        |     # rotate 180 degrees about x. then rotate (90 deg + heading1 degrees) about z ccw
        |     m1 = get_rotation_matrix_from_description("x", -1, 180 * pi / 180)
        |     m2 = get_rotation_matrix_from_description("z", 1, heading1 + pi/2)
        |     m3 = multiply_matrix(m2, m1) #we rotate m1 first then m2, so we multiply in backwards order: 2 then 1
        |     rxryrz2 = convert_matrix_to_axang(m3)
        |     rx2 = rxryrz2[0]
        |     ry2 = rxryrz2[1]
        |     rz2 = rxryrz2[2]
        | 
        |     # calculate point centerchamfers (where the center of the two chamfers intersect
        |     pcx = x0 + (leftwallthickmm + deepchambumpmm) * l1delxunit + (rightwallthickmm + deepchambumpmm) * l2delxunit
        |     pcy = y0 + (leftwallthickmm + deepchambumpmm) * l1delyunit + (rightwallthickmm + deepchambumpmm) * l2delyunit
        |     pcz = z0
        | 
        |     # calculate point1 (start of weld)
        |     p1x = pcx + l2delxunit * wd1
        |     p1y = pcy + l2delyunit * wd1
        |     p1z = pcz
        |     point1 = p[p1x, p1y, p1z, rx1, ry1, rz1]
        | 
        |     # calculate point2 (end of segment 1)
        |     p2x = pcx
        |     p2y = pcy
        |     p2z = pcz
        |     point2 = p[p2x, p2y, p2z, rx1, ry1, rz1]
        | 
        |     # calculate point3 (point at end of turn)
        |     slide = 0.00 # slide distance : the distance the tip slides forward as it turns
        |     p3x = pcx + slide * l1delxunit
        |     p3y = pcy + slide * l1delyunit
        |     p3z = pcz
        |     point3 = p[p3x, p3y, p3z, rx2, ry2, rz2]
        | 
        |     # calculate point4 (end of segment 2)
        |     p4x = pcx + wd2 * l1delxunit
        |     p4y = pcy + wd2 * l1delyunit
        |     p4z = pcz
        |     point4 = p[p4x, p4y, p4z, rx2, ry2, rz2]
        | 
        |     # third path
        | 
        |     # calculate rxryrz3 (gun pointing down, preheat pointing toward corner. for right seam, pointing right)
        |     # start with rxryrz = 0,0,0 (gun facing up, preheat facing y+ axis.
        |     # rotate it 180 degrees about x axis. gun facing down, preheat facing y- axis
        |     # rotate it about 135 degrees ccw about z axis. x+ to heading3 is about 225 degrees. so our angle is heading3 - 90 degrees
        |     m1 = get_rotation_matrix_from_description("x", -1, 180 * pi / 180) # rotation 1: 180 degrees forward about x axis
        |     m2 = get_rotation_matrix_from_description("z", 1, heading3 - pi/2) # rotation 2
        |     m3 = multiply_matrix(m2, m1) #we rotate m1 first then m2, so we multiply in backwards order: 2 then 1
        |     rxryrz3 = convert_matrix_to_axang(m3)
        |     rx3 = rxryrz3[0]
        |     ry3 = rxryrz3[1]
        |     rz3 = rxryrz3[2]
        | 
        |     # calculate rxryrz4 (gun at 45 around corner)
        |     m1 = get_rotation_matrix_from_description("x", -1, 135 * pi / 180) # rotation 1: 135 degrees forward about x axis
        |     m2 = get_rotation_matrix_from_description("z", 1, heading3 - pi/2)
        |     m3 = multiply_matrix(m2, m1) #we rotate m1 first then m2, so we multiply in backwards order: 2 then 1
        |     rxryrz4 = convert_matrix_to_axang(m3)
        |     rx4 = rxryrz4[0]
        |     ry4 = rxryrz4[1]
        |     rz4 = rxryrz4[2]
        | 
        |     # calculate rxryrz5 (gun straight into right seam side chamfer, preheat down)
        |     # rotate about x 90 (forward). then rotate about z ~ 135 (ccw)
        |     m1 = get_rotation_matrix_from_description("x", -1, 90 * pi / 180)
        |     m2 = get_rotation_matrix_from_description("z", 1, heading3 - pi/2)
        |     m3 = multiply_matrix(m2, m1) #we rotate m1 first then m2, so we multiply in backwards order: 2 then 1
        |     rxryrz5 = convert_matrix_to_axang(m3)
        |     rx5 = rxryrz5[0]
        |     ry5 = rxryrz5[1]
        |     rz5 = rxryrz5[2]
        | 
        |     # calculate rxryrz6 (gun straight into right seam side chamfer, preheat down, 10 degrees tiltback)
        |     tiltangledeg = 10 # ten degree angle of tilt
        |     m1 = get_rotation_matrix_from_description("x", -1, (90 + tiltangledeg) * pi / 180) # rotation 1: 135 degrees forward about x axis
        |     m2 = get_rotation_matrix_from_description("z", 1, heading3 - pi/2)
        |     m3 = multiply_matrix(m2, m1) #we rotate m1 first then m2, so we multiply in backwards order: 2 then 1
        |     rxryrz6 = convert_matrix_to_axang(m3)
        |     rx6 = rxryrz6[0]
        |     ry6 = rxryrz6[1]
        |     rz6 = rxryrz6[2]
        | 
        |     # calculate pointtopcham (the point at the top of the endwall chamfer) ( WHERE POINT3 WOULD BE IF RADIUS WAS 0)
        |     ptcx = x0 + leftwallthickmm * l1delxunit
        |     ptcy = y0 + leftwallthickmm * l1delyunit
        |     ptcz = z0
        | 
        |     # calculate point201 (weld start)
        |     # if deepchamfer, just ignore that. because if its deep chamfer then it filled more as well. so the hot extrudant should be to the same spot (same distance from the pointtopcham) whether it's big weld or small weld
        |     adjust = 0.0 # if you want to move the start point further away from corner (positive, mm) or closer to corner
        |     p201x = x0 + rightwallthickmm * l2delxunit + leftwallthickmm * l1delxunit + adjust * l2delxunit
        |     p201y = y0 + rightwallthickmm * l2delyunit + leftwallthickmm * l1delyunit + adjust * l2delyunit
        |     p201z = z0
        |     point201 = p[p201x, p201y, p201z, rx3, ry3, rz3]
        | 
        |     # the round over distance is the distance from pointbottomvcham to point2 (which will be the same as distance to p4)
        |     roundoverdistance = 0.05
        |     rod = roundoverdistance * 25.4 / 1000
        | 
        |     # calculate point202 (start of roundover)
        |     p202x = ptcx + rod * l2delxunit
        |     p202y = ptcy + rod * l2delyunit
        |     p202z = z0
        |     point202 = p[p202x, p202y, p202z, rx3, ry3, rz3]
        | 
        |     # calculate point203 (middle of roundover)
        |     # we know that the angle is exactly 90 degrees
        |     delta = calc_rod_midpoint_90deg(rod)
        |     p203z = ptcz - delta
        |     p203x = ptcx + delta * l2delxunit
        |     p203y = ptcy + delta * l2delyunit
        |     point203 = p[p203x, p203y, p203z, rx4, ry4, rz4]
        | 
        |     # calculate point204 (end of roundover)
        |     point204 = p[ptcx, ptcy, ptcz - rod, rx5, ry5, rz5]
        | 
        |     # calculate trail out points (tilt back and ride)
        |     botvcham = wd3 # where is the bottom of the v chamfer (z distance from top corner)
        |     tcpdiff = 14 # mm. the difference between backofhole tcp and welder tcp (tip)
        |     # point101 will still use backofhole, but points 102 and 103 will use normal weld tip tcp
        |     # calculate point5a (point101) (start of tilt back) (start of unflatten)
        |     dist = 1.5 * 25.4/1000 + tcpdiff/1000 # distance from botvcham
        |     p101x = ptcx
        |     p101y = ptcy
        |     p101z = ptcz - wd3 + dist
        |     point101 = p[p101x, p101y, p101z, rx5, ry5, rz5]
        | 
        |     # calculate point5b (point 102) (end of unflatten)
        |     dist = 0.5 * 25.4 / 1000
        |     tiltraise = 0.006
        |     p102x = ptcx + l2delxunit * tiltraise * -1
        |     p102y = ptcy + l2delyunit * tiltraise * -1
        |     p102z = ptcz - wd3 + dist
        |     point102 = p[p102x, p102y, p102z, rx6, ry6, rz6]
        | 
        |     # calculate point 5c (point 103) (end of smear)
        |     dist = -2 * 25.4/1000
        |     point103 = p[p102x, p102y, ptcz - wd3 + dist, rx6, ry6, rz6]
        | 
        |     # return
        |     struct2 = struct(point1=point1, point2=point2, point3=point3, point4=point4, point201=point201, point202=point202, point203=point203, point204=point204, point101=point101, point102=point102, point103=point103)
        |     return struct2
        | 
        | end
        | 
        | 
        | def main_calculate_cover_straight(p11, p12, p21, p22, sidewallthick, leftpoint, rightpoint, deepcovercham):
        |     struct1 = analyze_touchpoints_only_cover_straight(p11, p12, p21, p22, leftpoint)
        |     struct2 = calculate_straight_points_cover(struct1, sidewallthick, leftpoint, rightpoint, deepcovercham)
        |     #struct2 = calculate_DOtA_points_left_extended(struct1, list1, chamferover, chamferup, tcp_pose_top)
        |     #struct3 = check_validity_left(struct1, struct2)
        |     return struct2
        | 
        | end
        | 
        | # calculates the line of intersection of the sidewall plane (assumed vertical) and the cover plane (assumed perpendicular to sidewall plane)
        | # returns a struct containing point0 (point on the intersection line, same y as leftpoint) and 3 components of the unit vector left to right and 2 components of the other direction in 2d
        | def analyze_touchpoints_only_cover_straight(p11, p12, p21, p22, leftpoint):
        |     # calculate slope of sidewall in x-y plane
        |     # get the raw points from the first line
        |     l1p1x=p11[0]
        |     l1p1y=p11[1]
        |     l1p2x=p12[0]
        |     l1p2y=p12[1]
        | 
        |     # equate the first line in 2d space
        |     ml1 = (l1p2y-l1p1y) / (l1p2x-l1p1x)
        | 
        |     # b = y - mx
        |     bl1 = l1p1y - ml1 * l1p1x
        | 
        |     # calculate the cover plane
        |     # if two planes are perpendicular, then their normal vectors must be perpendicular.
        |     # the first planes normal vector is n1, which is taken from the equation of the plane ax + by + cz = d -> <a, b, c>
        |     # the second plane's normal vector is perpendicular to all vectors contained in the plane
        |     # p21 to p22 is a vector v contained within plane 2.
        |     # n2 is normal to both n1 AND v. to achieve a vector that is normal to both, take the cross product
        | 
        |     # plane 1 (y = mx + b) -> (b = -mx +1y +0z)
        |     n1 = [-1 * ml1, 1, 0]
        | 
        |     # v=P2−P1=(x2−x1,y2−y1,z2−z1)
        |     v = [p21[0]-p22[0], p21[1]-p22[1], p21[2]-p22[2]]
        | 
        |     #v n2 = cross product of n1 and v
        |     n2x = n1[1]*v[2] - n1[2]*v[1]
        |     n2y = n1[2]*v[0] - n1[0]*v[2]
        |     n2z = n1[0]*v[1] - n1[1]*v[0]
        |     n2 = [n2x, n2y, n2z]
        | 
        |     # find the d of the second plane
        |     # n2x * x + n2y * y + n2z * z = d0
        |     d = n2x * p21[0] + n2y * p21[1] + n2z * p21[2]
        | 
        |     # find the intersection line of the two planes
        |     # find the direction vector of that line by taking the cross product of the normal vector of those two planes
        |     v3x = n1[1]*n2[2] - n1[2]*n2[1]
        |     v3y = n1[2]*n2[0] - n1[0]*n2[2]
        |     v3z = n1[0]*n2[1] - n1[1]*n2[0]
        |     v3 = [v3x, v3y, v3z]
        | 
        |     # normalize the vector so the magnitude is 1
        |     magnitude2 = v3x * v3x + v3y * v3y + v3z * v3z
        |     magnitude = sqrt(magnitude2)
        |     v3xunit = v3x/magnitude
        |     v3yunit = v3y/magnitude
        |     v3zunit = v3z/magnitude
        | 
        |     # make sure it is going the right way (from left to right). make sure the v3yunit is positive
        |     if v3yunit < 0:
        |         v3xunit = v3xunit * -1
        |         v3yunit = v3yunit * -1
        |         v3zunit = v3zunit * -1
        |     end
        | 
        |     # next we have to find a point on the line by setting one of the dimensions and solving the system of equations
        |     # i will pick the y value of the left teach point
        |     y = leftpoint[1]
        |     # plane 1: -ml1 * x + 1 * y + 0 * z = bl1
        |     # -ml1 * x = bl1 - y
        |     x = (bl1 - y)/ (-1 * ml1)
        |     # plane 2: d = n2x * x + n2y * y + n2z * z
        |     # (d - n2x * x - n2y * y) = n2z * z
        |     z = (d - n2x * x - n2y * y) / n2z
        | 
        |     # make point0 into a pose
        |     point0 = p[x, y, z, 0, 0, 0]
        | 
        |     # find heading of main line
        |     heading1 = convert_uv_to_heading(v3xunit, v3yunit)
        | 
        |     # make a unit vector perpendicular to this one in the xy plane pointing x -. will be used to move over the chamfer distance
        |     ml2 = -1 / ml1
        |     # y = ml2 * x + unknownB
        |     # vector = [1, ml2]
        |     mag2 = 1 + ml2 * ml2
        |     mag = sqrt(mag2)
        |     v4xunit = 1 / mag
        |     v4yunit = ml2 / mag
        |     # switch is to the x direction is negative
        |     v4xunit = -1 * v4xunit
        |     v4yunit = -1 * v4yunit
        | 
        |     ret = struct(point0=point0, v3xunit=v3xunit, v3yunit=v3yunit, v3zunit=v3zunit, heading1=heading1, v4xunit=v4xunit, v4yunit=v4yunit)
        |     return ret
        | end
        | 
        | def calculate_straight_points_cover(struct1, sidewallthick, leftpointteach, rightpointteach, deepcovercham):
        |     # get the stuff
        |     point0 = struct1[0]
        |     p0x = point0[0]
        |     p0y = point0[1]
        |     p0z = point0[2]
        |     v3xunit = struct1[1]
        |     v3yunit = struct1[2]
        |     v3zunit = struct1[3]
        |     heading1 = struct1[4]
        |     v4xunit = struct1[5]
        |     v4yunit = struct1[6]
        |     sidewallthick = sidewallthick
        |     lpy = leftpointteach[1]
        |     rpy = rightpointteach[1]
        | 
        |     # first, check if we need a lift column raise
        |     # (we do, because for maximum reach we want to make the lift pedestal be even with the top of the covers)
        |     zpi = p0z
        |     if zpi > 0:
        |         liftcolumnzneeded = zpi * 1000.0 # the robot uses coordinates in meters, but the lift column uses coordinates in mm
        |         coverz = 0
        |     else:
        |         coverz = zpi
        |     end
        | 
        |     if deepcovercham:
        |         deepchambumpmm = 0.09 * 25.4/1000 # if there is a deep chamfer on the cover, bump the welder inwards 0.09 more inches.
        |     else:
        |         deepchambumpmm = 0.0
        |     end
        | 
        |     # calculate pointtopvcham
        |     chamferover = sidewallthick * 25.4 / 1000.0 + deepchambumpmm
        |     tiltraise = 0.006 # 6 mm raise needed for the tip to clear the plane during tiltback
        |     x = p0x + v4xunit * chamferover
        |     y = p0y + v4yunit * chamferover
        |     z = coverz + tiltraise
        | 
        |     # calculate rxryrz for tilted back
        |     # 3 rotations to make this happen.
        |     # start point is straight up with the preheat pointed in the +y direction.
        |     # first rotation is 180 degrees about x direction. gun is now pointing straight down with preheat facing -y direction
        |     m1 = get_rotation_matrix_from_description("x", 1, 180 * pi / 180)
        |     # second rotation is a 10 degree turn about the x axis (negative direction)
        |     m2 = get_rotation_matrix_from_description("x", -1, 10 * pi / 180)
        |     # third rotation is about 180 degrees about the z axis. starting from the -y axis, go until you get to heading1. that will equal heading1 plus 90 degrees
        |     m3 = get_rotation_matrix_from_description("z", 1, pi/2 + heading1)
        |     # combine them by multiplying m3 * m2 * m1
        |     # matrix multiplication is not commutative but it IS associative, so you can do this whichever order
        |     m4 = multiply_matrix(m2, m1)
        |     m5 = multiply_matrix(m3, m4)
        |     rxryrzt = convert_matrix_to_axang(m5)
        |     rxt = rxryrzt[0]
        |     ryt = rxryrzt[1]
        |     rzt = rxryrzt[2]
        |     pointtopvcham = p[x, y, z, rxt, ryt, rzt]
        | 
        |     # calculate point1 (preheat)
        |     dist = -1 * 25.4 / 1000.0 # move back 1 inch from
        |     p1x = x + dist * v3xunit
        |     p1y = y + dist * v3yunit
        |     p1z = z + dist * v3zunit
        |     point1 = p[p1x, p1y, p1z, rxt, ryt, rzt]
        | 
        |     # calculate point2 (start of flatten)
        |     dist = 0.5 * 25.4 / 1000.0  # half an inch past the top of v chamfer
        |     p2x = x + dist * v3xunit
        |     p2y = y + dist * v3yunit
        |     p2z = z + dist * v3zunit
        |     point2 = p[p2x, p2y, p2z, rxt, ryt, rzt]
        | 
        |     # calculate rxryrz for nontilted
        |     # first rotation is 180 degrees about x direction. gun is now pointing straight down with preheat facing -y direction
        |     m1 = get_rotation_matrix_from_description("x", 1, 180 * pi / 180)
        |     # third rotation is about 180 degrees about the z axis. starting from the -y axis, go until you get to heading1. that will equal heading1 plus 90 degrees
        |     m3 = get_rotation_matrix_from_description("z", 1, pi/2 + heading1)
        |     m5 = multiply_matrix(m3, m1)
        |     rxryrz = convert_matrix_to_axang(m5)
        |     rx = rxryrz[0]
        |     ry = rxryrz[1]
        |     rz = rxryrz[2]
        | 
        |     # calculate point3 (end of flatten)
        |     dist = 1.5 * 25.4 / 1000.0  # 1.5 inches past top of v chamfer
        |     p3x = x + dist * v3xunit
        |     p3y = y + dist * v3yunit
        |     p3z = coverz + dist * v3zunit
        |     point3 = p[p3x, p3y, p3z, rx, ry, rz]
        | 
        |     # calculate distance between leftpoint and rightpoint
        |     # we have the y distance. we need to find the total distance.
        |     # the unit vector (v3) should have a magnitude of 1. that's what analyze_touchpoints_only_cover_straight() calculated.
        |     # so the total distance is y distance * 1 / v3yunit
        |     ydist = rpy - lpy
        |     totdist = ydist / v3yunit
        | 
        |     # calculate pointtopvcham2
        |     x2 = x + v3xunit * totdist
        |     y2 = y + v3yunit * totdist
        |     z2 = z + v3zunit * totdist
        | 
        |     # calculate point4 (start of unflatten)
        |     dist = -1.5 * 25.4 / 1000.0
        |     p4x = x2 + v3xunit * dist
        |     p4y = y2 + v3yunit * dist
        |     p4z = z2 + v3zunit * dist - tiltraise
        |     point4 = p[p4x, p4y, p4z, rx, ry, rz]
        | 
        |     # calculate point5 (end of unflatten)
        |     dist = -0.5 * 25.4 / 1000.0
        |     p5x = x2 + v3xunit * dist
        |     p5y = y2 + v3yunit * dist
        |     p5z = z2 + v3zunit * dist
        |     point5 = p[p5x, p5y, p5z, rxt, ryt, rzt]
        | 
        |     # calculate point6 (end of smear)
        |     dist = 2 * 25.4 / 1000.0
        |     p6x = x2 + v3xunit * dist
        |     p6y = y2 + v3yunit * dist
        |     p6z = z2 + v3zunit * dist
        |     point6 = p[p6x, p6y, p6z, rxt, ryt, rzt]
        | 
        | 
        |     # return struct
        |     ret = struct(pointtopvcham=pointtopvcham, point1=point1, point2=point2, point3=point3, point4=point4, point5=point5, point6=point6)
        |     return ret
        | 
        | 
        | end
        | 
        | def main_calculate_floor_straight(p11, p12, p21, p22, floorthick, leftpoint, rightpoint):
        |     struct1 = analyze_touchpoints_only_cover_straight(p11, p12, p21, p22, leftpoint)
        |     struct2 = calculate_straight_points_floor(struct1, floorthick, leftpoint, rightpoint)
        |     #struct2 = calculate_DOtA_points_left_extended(struct1, list1, chamferover, chamferup, tcp_pose_top)
        |     #struct3 = check_validity_left(struct1, struct2)
        |     return struct2
        | 
        | end
        | 
        | # the path for welding a floor straight weld with v chisels on both sides.
        | # start at the right side and move left.
        | def calculate_straight_points_floor(struct1, floorthick, leftpointteach, rightpointteach):
        |     # get the stuff
        |     point0 = struct1[0]
        |     p0x = point0[0]
        |     p0y = point0[1]
        |     p0z = point0[2]
        |     v3xunit = struct1[1]
        |     v3yunit = struct1[2]
        |     v3zunit = struct1[3]
        |     heading1 = struct1[4]
        |     v4xunit = struct1[5]
        |     v4yunit = struct1[6]
        |     lpy = leftpointteach[1]
        |     rpy = rightpointteach[1]
        | 
        |     # first, check if we need a lift column raise
        |     # (we do not, because the floors are low)
        |     zpi = p0z
        |     floorz = zpi
        | 
        |     # calculate pointtopvcham (left point) (tilted and tiltraised)
        |     chamferup = floorthick * 25.4 / 1000.0
        |     tiltraise = 0.006 # 6 mm raise needed for the tip to clear the plane during tiltback
        |     # on this one, move the tiltraise distance sideways (towards robot) and the chamferover distance up
        |     x = p0x + v4xunit * tiltraise * -1
        |     y = p0y + v4yunit * tiltraise * -1
        |     z = floorz + chamferup
        | 
        |     # calculate rxryrz for tilted back
        |     # 3 rotations to make this happen.
        |     # start point is straight up with the preheat pointed in the +y direction.
        |     # first rotation is 90 degrees about y axis. positive direction. gun is now pointing in the x+ direction with preheat facing +y direction
        |     m1 = get_rotation_matrix_from_description("y", 1, 90 * pi / 180)
        |     # second rotation is about 180 degrees about the z axis. heading1 plus 90 degrees. gun is now pointing directly into the sidewall
        |     m2 = get_rotation_matrix_from_description("z", 1, pi/2 + heading1)
        |     # third rotation is 10 degrees about the z axis. gun is now tilted back 10 degrees from the sidewall
        |     m3 = get_rotation_matrix_from_description("z", 1, 10 * pi / 180)
        |     # combine them by multiplying m3 * m2 * m1
        |     # matrix multiplication is not commutative but it IS associative, so you can do this whichever order
        |     m4 = multiply_matrix(m2, m1)
        |     m5 = multiply_matrix(m3, m4)
        |     rxryrzt = convert_matrix_to_axang(m5)
        |     rxt = rxryrzt[0]
        |     ryt = rxryrzt[1]
        |     rzt = rxryrzt[2]
        |     # the non tilted angle is just m4
        |     rxryrz = convert_matrix_to_axang(m4)
        |     rx = rxryrz[0]
        |     ry = rxryrz[1]
        |     rz = rxryrz[2]
        |     pointtopvcham = p[x, y, z, rxt, ryt, rzt]
        | 
        |     # calculate distance between leftpoint and rightpoint
        |     # we have the y distance. we need to find the total distance.
        |     # the unit vector (v3) should have a magnitude of 1. that's what analyze_touchpoints_only_cover_straight() calculated.
        |     # so the total distance is y distance * 1 / v3yunit
        |     ydist = rpy - lpy
        |     totdist = ydist / v3yunit
        | 
        |     # calculate pointtopvcham2 (right point) (tilted and tiltraised)
        |     x2 = x + v3xunit * totdist
        |     y2 = y + v3yunit * totdist
        |     z2 = z + v3zunit * totdist
        |     pointtopvcham2 = p[x2, y2, z2, rxt, ryt, rzt]
        | 
        |     # calculate point1 (preheat)
        |     dist = 1 * 25.4 / 1000.0 # move back 1 inch from ptvc2 (in this case back means positive)
        |     p1x = x2 + dist * v3xunit
        |     p1y = y2 + dist * v3yunit
        |     p1z = z2 + dist * v3zunit
        |     point1 = p[p1x, p1y, p1z, rxt, ryt, rzt]
        | 
        |     # calculate point2 (start of flatten)
        |     dist = -0.5 * 25.4 / 1000.0  # half an inch past the top of v chamfer
        |     p2x = x2 + dist * v3xunit
        |     p2y = y2 + dist * v3yunit
        |     p2z = z2 + dist * v3zunit
        |     point2 = p[p2x, p2y, p2z, rxt, ryt, rzt]
        | 
        |     # calculate point3 (end of flatten)
        |     dist = -1.5 * 25.4 / 1000.0  # 1.5 inches past top of v chamfer
        |     p3x = x2 + dist * v3xunit + tiltraise * v4xunit
        |     p3y = y2 + dist * v3yunit + tiltraise * v4yunit
        |     p3z = z2 + dist * v3zunit
        |     point3 = p[p3x, p3y, p3z, rx, ry, rz]
        | 
        |     # calculate point4 (start of unflatten)
        |     dist = 1.5 * 25.4 / 1000.0
        |     p4x = x + v3xunit * dist + tiltraise * v4xunit
        |     p4y = y + v3yunit * dist + tiltraise * v4yunit
        |     p4z = z + v3zunit * dist
        |     point4 = p[p4x, p4y, p4z, rx, ry, rz]
        | 
        |     # calculate point5 (end of unflatten)
        |     dist = 0.5 * 25.4 / 1000.0
        |     p5x = x + v3xunit * dist
        |     p5y = y + v3yunit * dist
        |     p5z = z + v3zunit * dist
        |     point5 = p[p5x, p5y, p5z, rxt, ryt, rzt]
        | 
        |     # calculate point6 (end of smear)
        |     dist = -2 * 25.4 / 1000.0
        |     p6x = x + v3xunit * dist
        |     p6y = y + v3yunit * dist
        |     p6z = z + v3zunit * dist
        |     point6 = p[p6x, p6y, p6z, rxt, ryt, rzt]
        | 
        |     # return struct
        |     ret = struct(pointtopvcham=pointtopvcham, point1=point1, point2=point2, point3=point3, point4=point4, point5=point5, point6=point6)
        |     return ret
        | 
        | end
        | 
        | # this function determines the starting touchpoints for homing in on cover lt geometry
        | # includes two points above the cover lt, closer to the robot than the lt, facing down
        | def get_coverlt_homing_pathpoints(leftpoint, rightpoint):
        |     # get the teach position points
        |     lpx = leftpoint[0]
        |     lpy = leftpoint[1]
        |     lpz = leftpoint[2]
        |     rpx = rightpoint[0]
        |     rpy = rightpoint[1]
        |     rpz = rightpoint[2]
        | 
        |     # specify the distances from (in meters)
        |     d0 = 0.05 # how far from the cover to approach from
        |     d1 = 0.03 # how far the touchpints are pushed closer to the robot
        |     d2 = 0.00 # how far inwards the touchpoints are pushed
        | 
        |     # rxryrz
        |     rxryrz = [0.334, 3.124, 0]
        |     rx = rxryrz[0]
        |     ry = rxryrz[1]
        |     rz = rxryrz[2]
        | 
        |     # calculate the points
        |     ph1 = p[lpx + d1, lpy + d2, lpz + d0, rx, ry, rz] # left side approach
        |     ph2 = p[rpx + d1, rpy - d2, rpz + d0, rx, ry, rz] # right side approach
        | 
        |     ret = struct(ph1=ph1, ph2=ph2)
        |     is_robot_at_reachable_spot(leftpoint, ret)
        |     return ret
        | end
        | 
        | def main_calculate_cover_lt(p11, p12, leftpoint, rightpoint):
        |     struct1 = analyze_touchpoints_only_cover_lt(p11, p12, leftpoint, rightpoint)
        |     struct2 = calculate_points_cover_lt(struct1)
        |     #struct2 = calculate_DOtA_points_left_extended(struct1, list1, chamferover, chamferup, tcp_pose_top)
        |     #struct3 = check_validity_left(struct1, struct2)
        |     return struct2
        | 
        | end
        | 
        | def analyze_touchpoints_only_cover_lt(p11, p12, leftpoint, rightpoint):
        |     # calculate the slope of the groove in xy plane
        |     l1p1x = leftpoint[0]
        |     l1p1y = leftpoint[1]
        |     l1p2x = rightpoint[0]
        |     l1p2y = rightpoint[1]
        | 
        |     # equate the first line in 2d space
        |     ml1 = (l1p2y-l1p1y) / (l1p2x-l1p1x)
        | 
        |     # b = y - mx
        |     bl1 = l1p1y - ml1 * l1p1x
        | 
        |     # zraise (how much the z value changes from left point to right point
        |     zraise = p12[2] - p11[2]
        | 
        |     #get the calcpoints
        |     leftcalcpoint = [leftpoint[0], leftpoint[1], p11[2]]
        |     rightcalcpoint = [rightpoint[0], rightpoint[1], p12[2]]
        |     # get the vector from a to b
        |     vec = [rightcalcpoint[0] - leftcalcpoint[0], rightcalcpoint[1] - leftcalcpoint[1], rightcalcpoint[2] - leftcalcpoint[2]]
        |     # get the unit vector in 3d
        |     mag3d = sqrt(vec[0]*vec[0]+vec[1]*vec[1]+vec[2]*vec[2])
        |     vec3dunit = [vec[0]/mag3d, vec[1]/mag3d, vec[2]/mag3d]
        |     # get the unit vector in 2d
        |     mag2d = sqrt(vec[0]*vec[0]+vec[1]*vec[1])
        |     vec2dunit = [vec[0]/mag2d, vec[1]/mag2d]
        |     # get the heading
        |     heading1 = convert_uv_to_heading(vec2dunit[0], vec2dunit[1])
        | 
        |     ret = struct(leftcalcpoint=leftcalcpoint, rightcalcpoint=rightcalcpoint, vxunit=vec3dunit[0], vyunit=vec3dunit[1], vzunit=vec3dunit[2], heading1=heading1)
        |     return ret
        | end
        | 
        | def calculate_points_cover_lt(struct1):
        |     # get the stuff from struct
        |     leftcalcpoint = struct1[0]
        |     x = leftcalcpoint[0]
        |     y = leftcalcpoint[1]
        |     z = leftcalcpoint[2]
        |     rightcalcpoint = struct1[1]
        |     x2 = rightcalcpoint[0]
        |     y2 = rightcalcpoint[1]
        |     z2 = rightcalcpoint[2]
        |     v3xunit = struct1[2]
        |     v3yunit = struct1[3]
        |     v3zunit = struct1[4]
        |     heading1 = struct1[5]
        | 
        |     # first calculate rxryrz f normal and tiltback
        |     # calculate rxryrz for tilted back
        |     # 3 rotations to make this happen.
        |     # start point is straight up with the preheat pointed in the +y direction.
        |     # first rotation is 180 degrees about x direction. gun is now pointing straight down with preheat facing -y direction
        |     m1 = get_rotation_matrix_from_description("x", 1, 180 * pi / 180)
        |     # second rotation is a 10 degree turn about the x axis (negative direction)
        |     m2 = get_rotation_matrix_from_description("x", -1, 10 * pi / 180)
        |     # third rotation is about 180 degrees about the z axis. starting from the -y axis, go until you get to heading1. that will equal heading1 plus 90 degrees
        |     m3 = get_rotation_matrix_from_description("z", 1, pi/2 + heading1)
        |     # combine them by multiplying m3 * m2 * m1
        |     # matrix multiplication is not commutative but it IS associative, so you can do this whichever order
        |     m4 = multiply_matrix(m2, m1)
        |     m5 = multiply_matrix(m3, m4)
        |     rxryrzt = convert_matrix_to_axang(m5)
        |     rxt = rxryrzt[0]
        |     ryt = rxryrzt[1]
        |     rzt = rxryrzt[2]
        | 
        |     # calculate rxryrz for nontilted
        |     # first rotation is 180 degrees about x direction. gun is now pointing straight down with preheat facing -y direction
        |     m1 = get_rotation_matrix_from_description("x", 1, 180 * pi / 180)
        |     # third rotation is about 180 degrees about the z axis. starting from the -y axis, go until you get to heading1. that will equal heading1 plus 90 degrees
        |     m3 = get_rotation_matrix_from_description("z", 1, pi/2 + heading1)
        |     m5 = multiply_matrix(m3, m1)
        |     rxryrz = convert_matrix_to_axang(m5)
        |     rx = rxryrz[0]
        |     ry = rxryrz[1]
        |     rz = rxryrz[2]
        | 
        |     tiltraise = 0.006 # 6 mm raise needed for the tip to clear the plane during tiltback
        | 
        |     # calculate points 1-3
        |     # calculate point1 (preheat)
        |     dist = -1 * 25.4 / 1000.0 # move back 1 inch from
        |     p1x = x + dist * v3xunit
        |     p1y = y + dist * v3yunit
        |     p1z = z + dist * v3zunit + tiltraise
        |     point1 = p[p1x, p1y, p1z, rxt, ryt, rzt]
        | 
        |     # calculate point2 (start of flatten)
        |     dist = 0.5 * 25.4 / 1000.0  # half an inch past the top of v chamfer
        |     p2x = x + dist * v3xunit
        |     p2y = y + dist * v3yunit
        |     p2z = z + dist * v3zunit + tiltraise
        |     point2 = p[p2x, p2y, p2z, rxt, ryt, rzt]
        | 
        |     # calculate point3 (end of flatten)
        |     dist = 1.5 * 25.4 / 1000.0  # 1.5 inches past top of v chamfer
        |     p3x = x + dist * v3xunit
        |     p3y = y + dist * v3yunit
        |     p3z = z + dist * v3zunit
        |     point3 = p[p3x, p3y, p3z, rx, ry, rz]
        | 
        |     # calculate points 4-6
        |     # calculate point4 (start of unflatten)
        |     dist = -1.5 * 25.4 / 1000.0
        |     p4x = x2 + v3xunit * dist
        |     p4y = y2 + v3yunit * dist
        |     p4z = z2 + v3zunit * dist
        |     point4 = p[p4x, p4y, p4z, rx, ry, rz]
        | 
        |     # calculate point5 (end of unflatten)
        |     dist = -0.5 * 25.4 / 1000.0
        |     p5x = x2 + v3xunit * dist
        |     p5y = y2 + v3yunit * dist
        |     p5z = z2 + v3zunit * dist + tiltraise
        |     point5 = p[p5x, p5y, p5z, rxt, ryt, rzt]
        | 
        |     # calculate point6 (end of smear)
        |     dist = 2 * 25.4 / 1000.0
        |     p6x = x2 + v3xunit * dist
        |     p6y = y2 + v3yunit * dist
        |     p6z = z2 + v3zunit * dist + tiltraise
        |     point6 = p[p6x, p6y, p6z, rxt, ryt, rzt]
        | 
        |     # return struct
        |     ret = struct(pointtopvcham=leftcalcpoint, point1=point1, point2=point2, point3=point3, point4=point4, point5=point5, point6=point6)
        |     return ret
        | 
        | end
        | 
        | def main_calculate_sleeve_fillet(p1, p2, p3):
        |     struct1 = analyze_touchpoints_only_sleeve_fillet(p1, p2, p3)
        |     struct2 = calculate_points_sleeve_fillet_quadonly(struct1)
        |     return struct2
        | end
        | 
        | # given 3 points at the intersection of the sleeve and the sidewall, this calculates and returns 3 things:
        | # the centerpoint of the circle on the plane, the normal vector of the plane, and the radius of the circle
        | # then it returns 4 more things after converting to a vertical circle/plane: heading1 (into the plane), vecn, vecr, vecu
        | def analyze_touchpoints_only_sleeve_fillet(p1, p2, p3):
        |     x1 = p1[0]
        |     y1 = p1[1]
        |     z1 = p1[2]
        |     x2 = p2[0]
        |     y2 = p2[1]
        |     z2 = p2[2]
        |     x3 = p3[0]
        |     y3 = p3[1]
        |     z3 = p3[2]
        | 
        |     # calculate plane
        |     # calculate ab (1->2) vector
        |     abvec = [x2-x1, y2-y1, z2-z1]
        |     # calculate ac (1->3) vector
        |     acvec = [x3-x1, y3-y1, z3-z1]
        |     #calculate the plane's normal vector = ab x ac
        | 
        |     n = crossproduct(abvec, acvec)
        |     mag = sqrt(n[0]*n[0]+n[1]*n[1]+n[2]*n[2])
        |     n = [n[0]/mag, n[1]/mag, n[2]/mag]
        |     d = n[0] * x1 + n[1] * y1 + n[2] * z1
        | 
        |     # find the circle
        |     # Midpoint of AB:
        |     mab = [(x1 + x2)/2, (y1 + y2)/2, (z1 + z2)/2]
        |     # midpoint of ac
        |     mac = [(x3 + x1)/2, (y3 + y1)/2, (z3 + z1)/2]
        |     # Get Normal Vectors to AB and AC in the Plane
        |     # nab (normal to ab) = abvec x n
        |     nab = crossproduct(abvec, n)
        |     # nac (normal to ac) = acvec x n
        |     nac = crossproduct(acvec, n)
        |     # Define Perpendicular Bisector Lines
        |     # Each line goes through a midpoint and extends in the direction of the na_
        |     # we already have the equations of those lines in point vector form with l1 = mab + s * nab, and l2 = mac + t * nac
        |     # define all the terms so the math is simpler when i have to do math
        |     mabx = mab[0]
        |     maby = mab[1]
        |     mabz = mab[2]
        |     nabx = nab[0]
        |     naby = nab[1]
        |     nabz = nab[2]
        |     macx = mac[0]
        |     macy = mac[1]
        |     macz = mac[2]
        |     nacx = nac[0]
        |     nacy = nac[1]
        |     nacz = nac[2]
        |     # find the intersection point using the y and z equations
        |     # maby + s * naby = macy + t * nacy
        |     # mabz + s * nabz = macz + t * nacz
        |     # first solve for s and take
        |     # t = (macz*naby + maby*nabz - mabz*naby - macy*nabz) / (nacy*nabz - naby*nacz)
        |     t = (macz*naby + maby*nabz - mabz*naby - macy*nabz) / (nacy*nabz - naby*nacz)
        |     # s = (t*nacz + macz - mabz) / nabz
        |     s = (t*nacz + macz - mabz) / nabz
        |     # find the point
        |     # pcenter = mac + t * nac
        |     pcenterx = macx + t * nacx
        |     pcentery = macy + t * nacy
        |     pcenterz = macz + t * nacz
        |     rxryrz = [0.528, 4.631, 0.258] # demo point of the welder pointing forward into a sleeve
        |     pcenter = p[pcenterx, pcentery, pcenterz, rxryrz[0], rxryrz[1], rxryrz[2]]
        |     radius = distance_between(pcenterx, pcentery, pcenterz, x1, y1, z1)
        | 
        |     # ------ start calculation of vertical assumption -----
        |     # assume the plane close to vertical
        |     # fix it to make it actually vertical
        |     # calculate the unit vector of up, and the unit vector of right.
        |     # calculate the heading from the +x axis to pointing straight into the wall.
        |     # the unit vector of up is [0, 0, 1] (because the plane is verticalized) (for easier calculations)
        |     # first calculate the normal vector INTO the sidewall (make sure x is negative) and make it a unit vector
        |     vecn = [n[0], n[1], 0] # vector normal
        |     if vecn[0] > 0:
        |         vecn = [-n[0], -n[1], 0]
        |     end
        |     mag = sqrt(vecn[0]*vecn[0]+vecn[1]*vecn[1])
        |     vecn = [vecn[0]/mag, vecn[1]/mag, 0]
        |     # next calculate the right normal vector (the vector IN the plane that goes to the right)
        |     vecr = [vecn[1], -1*vecn[0], 0]
        |     vecu = [0, 0, 1] # vector up
        |     heading1 = convert_uv_to_heading(vecn[0], vecn[1])
        | 
        | 
        |     ret = struct(pcenter=pcenter, planenormalvec=n, radius=radius, heading1=heading1, vecn=vecn, vecr=vecr, vecu=vecu)
        |     return ret
        | end
        | 
        | def crossproduct(vec1, vec2):
        |     nx = vec1[1]*vec2[2] - vec1[2]*vec2[1]
        |     ny = vec1[2]*vec2[0] - vec1[0]*vec2[2]
        |     nz = vec1[0]*vec2[1] - vec1[1]*vec2[0]
        |     ret = [nx, ny, nz]
        |     return ret
        | end
        | 
        | def calculate_points_sleeve_fillet(struct1):
        | 
        | end
        | 
        | # this function calculates only the four points of the quadrants, for the not real program.
        | # these calculations are easier so that's why i'm starting with them first.
        | # this assumes a vertical plane
        | def calculate_points_sleeve_fillet_quadonly(struct1):
        |     # get the stuff from the struct
        |     pcenter = struct1[0]
        |     pcx = pcenter[0]
        |     pcy = pcenter[1]
        |     pcz = pcenter[2]
        |     planenormalvec = struct1[1]
        |     radius = struct1[2]
        |     heading1 = struct1[3]
        |     vecn = struct1[4]
        |     vecnx = vecn[0]
        |     vecny = vecn[1]
        |     vecr = struct1[5]
        |     vecrx = vecr[0]
        |     vecry = vecr[1]
        |     vecu = struct1[6]
        |     vecuz = vecu[2]
        | 
        |     # define cushions (the backofhole can't actually touch the intersection of pipe and wall, it travels a certain distance around it
        |     cushout = 0.006 # 5mm # the cushion out from the wall
        |     cusharound = 0.006 # 5mm # the cushion around the sleeve.
        | 
        |     # get the top point (point1)
        |     # take the center point and move up the radius plus the cushions
        |     p1x = pcx + vecnx * -1 * cushout
        |     p1y = pcy + vecny * -1 * cushout
        |     p1z = pcz + vecuz * radius + vecuz * cusharound
        | 
        |     # find rxryrz1
        |     # first rotation is 135 degrees about the y- direction. 90 degrees to get flat. Tip pointing x-, preheat pointing y+. 45 more degrees to get at that above angle
        |     m1 = get_rotation_matrix_from_description("y", -1, 135 * pi / 180)
        |     # second rotation is heading1 – 180 degrees about the z+ axis to get pointing straight into wall. Heading1 should be about 180 degrees
        |     m2 = get_rotation_matrix_from_description("z", 1, heading1 - 180 * pi/180)
        |     # combine them by multiplying
        |     m3 = multiply_matrix(m2, m1)
        |     rxryrz1 = convert_matrix_to_axang(m3)
        |     rx1 = rxryrz1[0]
        |     ry1 = rxryrz1[1]
        |     rz1 = rxryrz1[2]
        | 
        |     point1 = p[p1x, p1y, p1z, rx1, ry1, rz1]
        | 
        |     # get second point (right) (point2)
        |     # take the center point and move right the radius plus the cushions
        |     p2x = pcx + vecrx * radius + vecrx * cusharound + vecnx * -1 * cushout
        |     p2y = pcy + vecry * radius + vecry * cusharound + vecny * -1 * cushout
        |     p2z = pcz
        | 
        |     # find rxryrz2
        |     # first rotation is 90 degrees about the x- axis
        |     m1 = get_rotation_matrix_from_description("x", -1, 90 * pi / 180)
        |     # second rotation is About 135 degrees about the z+ axis. This calculation is heading1 – 45 degrees
        |     m2 = get_rotation_matrix_from_description("z", 1, heading1 - 45 * pi/180)
        |     # combine them by multiplying
        |     m3 = multiply_matrix(m2, m1)
        |     rxryrz2 = convert_matrix_to_axang(m3)
        |     rx2 = rxryrz2[0]
        |     ry2 = rxryrz2[1]
        |     rz2 = rxryrz2[2]
        | 
        |     point2 = p[p2x, p2y, p2z, rx2, ry2, rz2]
        | 
        |     # get the third point (bottom) (point3)
        |     p3x = pcx + vecnx * -1 * cushout
        |     p3y = pcy + vecny * -1 * cushout
        |     p3z = pcz - vecuz * radius - vecuz * cusharound
        | 
        |     # find rxryrz3
        |     # first rotation is 45 degrees about the y+ axis
        |     m1 = get_rotation_matrix_from_description("y", 1, 45 * pi / 180)
        |     # second rotation is About 180 degrees about the z+ axis. This calculation is heading1 degrees
        |     m2 = get_rotation_matrix_from_description("z", 1, heading1)
        |     # combine them by multiplying
        |     m3 = multiply_matrix(m2, m1)
        |     rxryrz3 = convert_matrix_to_axang(m3)
        |     rx3 = rxryrz3[0]
        |     ry3 = rxryrz3[1]
        |     rz3 = rxryrz3[2]
        | 
        |     point3 = p[p3x, p3y, p3z, rx3, ry3, rz3]
        | 
        |     # get the fourth point (left) (point4)
        |     p4x = pcx - vecrx * radius - vecrx * cusharound + vecnx * -1 * cushout
        |     p4y = pcy - vecry * radius - vecry * cusharound + vecny * -1 * cushout
        |     p4z = pcz
        | 
        |     # find rxryrz4
        |     # first rotation is 90 degrees about the x+ axis
        |     m1 = get_rotation_matrix_from_description("x", 1, 90 * pi / 180)
        |     # second rotation is heading1 + 45 degrees about the z+ axis. approx 225 degrees ccw
        |     m2 = get_rotation_matrix_from_description("z", 1, heading1 + 45 * pi/180)
        |     # combine them by multiplying
        |     m3 = multiply_matrix(m2, m1)
        |     rxryrz4 = convert_matrix_to_axang(m3)
        |     rx4 = rxryrz4[0]
        |     ry4 = rxryrz4[1]
        |     rz4 = rxryrz4[2]
        | 
        |     point4 = p[p4x, p4y, p4z, rx4, ry4, rz4]
        | 
        |     # return the points
        |     ret = struct(point1=point1, point2=point2, point3=point3, point4=point4)
        |     return ret
        | 
        | end
      tcp_pose_top := p[tp[0],tp[1],tp[2]+.2,tp[3],tp[4],tp[5]]
  path_pre := get_corner_homing_45_pathpoints(tp,tcp_pose_top)
  ph1 := path_pre[0]
  ph2 := path_pre[1]
  ph3 := path_pre[2]
  ph4 := path_pre[3]
  ph5 := path_pre[4]
  ph6 := path_pre[5]
  ph7 := path_pre[6]
  ph2up := path_pre[7]
  ph4up := path_pre[8]
  MoveL speed 250 mm/s, acceleration 200 mm/s^2 (useActiveTCP=true optimoveEnabled=false optiMoveSpeed=0.3 optiMoveAcceleration=0.09) feature=Base
    Waypoint Variable (Variable): variable=ph1
    Waypoint Variable (Variable): variable=ph2
  Wait Sleep waitTime=0.5
  MoveL speed 20 mm/s, acceleration 100 mm/s^2 (useActiveTCP=true optimoveEnabled=false optiMoveSpeed=0.3 optiMoveAcceleration=0.09) feature=Base
    MoveDirectionNode expression=[-1,-1.0,0.0]
      Until TOOL_CONTACT_DETECTION (allowActions=false retraction=0 decelerationAcceleration=3 decelerationAngularAcceleration=34.906585)
  p11 := get_actual_tcp_pose()
  MoveJ speed 60 deg/s, acceleration 80 deg/s^2 (useActiveTCP=true optimoveEnabled=false optiMoveSpeed=0.3 optiMoveAcceleration=0.09) feature=Base
    Waypoint Variable (Variable): variable=ph2
    Waypoint Variable (Variable): variable=ph2up
  Wait Sleep waitTime=0.5
  MoveL speed 20 mm/s, acceleration 100 mm/s^2 (useActiveTCP=true optimoveEnabled=false optiMoveSpeed=0.3 optiMoveAcceleration=0.09) feature=Base
    MoveDirectionNode expression=[-1,-1.0,0.0]
      Until TOOL_CONTACT_DETECTION (allowActions=false retraction=0 decelerationAcceleration=3 decelerationAngularAcceleration=34.906585)
  p13 := get_actual_tcp_pose()
  MoveJ speed 60 deg/s, acceleration 80 deg/s^2 (useActiveTCP=true optimoveEnabled=false optiMoveSpeed=0.3 optiMoveAcceleration=0.09) feature=Base
    Waypoint Variable (Variable): variable=ph2up
    Waypoint Variable (Variable): variable=ph3
  Wait Sleep waitTime=0.5
  MoveL speed 20 mm/s, acceleration 100 mm/s^2 (useActiveTCP=true optimoveEnabled=false optiMoveSpeed=0.3 optiMoveAcceleration=0.09) feature=Base
    MoveDirectionNode expression=[-1,-1.0,0.0]
      Until TOOL_CONTACT_DETECTION (allowActions=false retraction=0 decelerationAcceleration=3 decelerationAngularAcceleration=34.906585)
  p12 := get_actual_tcp_pose()
  SuppressedNode
    MoveJ speed 60 deg/s, acceleration 80 deg/s^2 (useActiveTCP=true optimoveEnabled=false optiMoveSpeed=0.3 optiMoveAcceleration=0.09) feature=Base
      Waypoint Variable (Variable): variable=ph3
      Waypoint Waypoint_4: TCP in base x=-658.265 y=299.53 z=30.91 mm, rx=0.4268 ry=-1.6215 rz=0.4371 rad; joints [-77.363, -55.591, 142.792, -102.186, -19.322, 105.94] deg; TCP offset x=0 y=0 z=246 mm, rx=0 ry=0 rz=0 rad
  MoveL speed 250 mm/s, acceleration 1200 mm/s^2 (useActiveTCP=true optimoveEnabled=false optiMoveSpeed=0.3 optiMoveAcceleration=0.09) feature=Base
    Waypoint Variable (Variable): variable=ph3
    Waypoint Variable (Variable): variable=ph1
  SuppressedNode
    MoveJ speed 60 deg/s, acceleration 80 deg/s^2 (useActiveTCP=true optimoveEnabled=false optiMoveSpeed=0.3 optiMoveAcceleration=0.09) feature=Base
      Waypoint Waypoint_5: TCP in base x=-448.863 y=524.6 z=-175.967 mm, rx=2.4733 ry=-1.8744 rz=0.2053 rad; joints [-65.056, -57.525, 139.86, -164.756, -91.924, 99.291] deg
      SuppressedNode
        Waypoint Waypoint_5: TCP in base x=-542.919 y=212.782 z=86.75 mm, rx=-0.746 ry=-1.5701 rz=-0.8083 rad; joints [-15.32, -63.738, 160.053, -88.648, -229.235, 89.501] deg
      Waypoint Waypoint_10: TCP in base x=-559.13 y=259.234 z=102.446 mm, rx=-0.8226 ry=-1.4861 rz=-0.8815 rad; joints [-31.871, -61.56, 166.811, -101.777, -239.831, 87.599] deg; TCP offset x=-1.157 y=-95.604 z=257.595 mm, rx=0 ry=0 rz=0 rad
  MoveL speed 250 mm/s, acceleration 1200 mm/s^2 (useActiveTCP=true optimoveEnabled=false optiMoveSpeed=0.3 optiMoveAcceleration=0.09) feature=Base
    Waypoint Variable (Variable): variable=ph4
  Wait Sleep waitTime=0.5
  MoveL speed 20 mm/s, acceleration 100 mm/s^2 (useActiveTCP=true optimoveEnabled=false optiMoveSpeed=0.3 optiMoveAcceleration=0.09) feature=Base
    MoveDirectionNode expression=[-1.0,1.0,0.0]
      Until TOOL_CONTACT_DETECTION (allowActions=false retraction=0 decelerationAcceleration=3 decelerationAngularAcceleration=34.906585)
  p21 := get_actual_tcp_pose()
  MoveL speed 250 mm/s, acceleration 1200 mm/s^2 (useActiveTCP=true optimoveEnabled=false optiMoveSpeed=0.3 optiMoveAcceleration=0.09) feature=Base
    Waypoint Variable (Variable): variable=ph4
    Waypoint Variable (Variable): variable=ph4up
  Wait Sleep waitTime=0.5
  MoveL speed 20 mm/s, acceleration 100 mm/s^2 (useActiveTCP=true optimoveEnabled=false optiMoveSpeed=0.3 optiMoveAcceleration=0.09) feature=Base
    MoveDirectionNode expression=[-1.0,1.0,0.0]
      Until TOOL_CONTACT_DETECTION (allowActions=false retraction=0 decelerationAcceleration=3 decelerationAngularAcceleration=34.906585)
  p23 := get_actual_tcp_pose()
  MoveL speed 250 mm/s, acceleration 1200 mm/s^2 (useActiveTCP=true optimoveEnabled=false optiMoveSpeed=0.3 optiMoveAcceleration=0.09) feature=Base
    Waypoint Variable (Variable): variable=ph4up
    Waypoint Variable (Variable): variable=ph5
  Wait Sleep waitTime=0.5
  MoveL speed 20 mm/s, acceleration 100 mm/s^2 (useActiveTCP=true optimoveEnabled=false optiMoveSpeed=0.3 optiMoveAcceleration=0.09) feature=Base
    MoveDirectionNode expression=[-1.0,1.0,0.0]
      Until TOOL_CONTACT_DETECTION (allowActions=false retraction=0 decelerationAcceleration=3 decelerationAngularAcceleration=34.906585)
  p22 := get_actual_tcp_pose()
  SuppressedNode
    MoveJ speed 60 deg/s, acceleration 80 deg/s^2 (useActiveTCP=true optimoveEnabled=false optiMoveSpeed=0.3 optiMoveAcceleration=0.09) feature=Base
      Waypoint Variable (Variable): variable=ph5
      Waypoint Variable (Variable): variable=ph4
      SuppressedNode
        Waypoint Waypoint_5: TCP in base x=-542.919 y=212.782 z=86.75 mm, rx=-0.746 ry=-1.5701 rz=-0.8083 rad; joints [-15.32, -63.738, 160.053, -88.648, -229.235, 89.501] deg; TCP offset x=0 y=0 z=246 mm, rx=0 ry=0 rz=0 rad
      Waypoint Waypoint_11: TCP in base x=-559.13 y=259.234 z=102.446 mm, rx=-0.8226 ry=-1.4861 rz=-0.8815 rad; joints [-31.871, -61.56, 166.811, -101.777, -239.831, 87.599] deg; TCP offset x=-1.157 y=-95.604 z=257.595 mm, rx=0 ry=0 rz=0 rad
      Waypoint Waypoint_12: TCP in base x=-448.863 y=524.6 z=-175.967 mm, rx=2.4733 ry=-1.8744 rz=0.2053 rad; joints [-65.056, -57.525, 139.86, -164.756, -91.924, 99.291] deg; TCP offset x=0 y=0 z=246 mm, rx=0 ry=0 rz=0 rad
      Waypoint Waypoint_4: TCP in base x=-658.265 y=299.53 z=30.91 mm, rx=0.4268 ry=-1.6215 rz=0.4371 rad; joints [-77.363, -55.591, 142.792, -102.186, -19.322, 105.94] deg
      Waypoint Waypoint_13: TCP in base x=-343.952 y=632.142 z=615.175 mm, rx=-0.0259 ry=-0.0088 rz=-0.5675 rad; joints [-77.363, -55.591, 142.791, -175.721, 90.298, 134.942] deg
      Waypoint Variable (Variable): variable=ph6
      Waypoint Variable (Variable): variable=ph7
  MoveJ speed 60 deg/s, acceleration 80 deg/s^2 (useActiveTCP=true optimoveEnabled=false optiMoveSpeed=0.3 optiMoveAcceleration=0.09) feature=Base
    Waypoint Variable (Variable): variable=ph5
  MoveL speed 250 mm/s, acceleration 1200 mm/s^2 (useActiveTCP=true optimoveEnabled=false optiMoveSpeed=0.3 optiMoveAcceleration=0.09) feature=Base
    Waypoint Variable (Variable): variable=ph4
    Waypoint Variable (Variable): variable=ph1
  MoveJ speed 60 deg/s, acceleration 80 deg/s^2 (useActiveTCP=true optimoveEnabled=false optiMoveSpeed=0.3 optiMoveAcceleration=0.09) feature=Base
    Waypoint Waypoint_4: TCP in base x=-658.265 y=299.53 z=30.91 mm, rx=0.4268 ry=-1.6215 rz=0.4371 rad; joints [-77.363, -55.591, 142.792, -102.186, -19.322, 105.94] deg
    Waypoint Waypoint_13: TCP in base x=-343.952 y=632.142 z=615.175 mm, rx=-0.0259 ry=-0.0088 rz=-0.5675 rad; joints [-77.363, -55.591, 142.791, -175.721, 90.298, 134.942] deg
    SuppressedNode
      Waypoint Waypoint_1: TCP in base x=-343.952 y=632.142 z=615.175 mm, rx=-0.025 ry=0.0331 rz=-3.0685 rad; joints [-76.965, -50.534, 141.988, -182.891, 90.622, -8.876] deg; TCP offset x=-0.345 y=-16.123 z=283.498 mm, rx=0 ry=0 rz=0 rad
    Waypoint Variable (Variable): variable=ph6
    Waypoint Variable (Variable): variable=ph7
  Wait Sleep waitTime=1
  SuppressedNode
    Folder debug
      MoveJ speed 60 deg/s, acceleration 80 deg/s^2 (useActiveTCP=true optimoveEnabled=false optiMoveSpeed=0.3 optiMoveAcceleration=0.09) feature=Base
        Waypoint ex_ph6: TCP in base x=-1187.196 y=387.122 z=-136.365 mm, rx=0 ry=0 rz=-3.1412 rad; joints [-26.656, 7.647, 65.2, -162.893, 89.928, -63.307] deg
  MoveL speed 20 mm/s, acceleration 100 mm/s^2 (useActiveTCP=true optimoveEnabled=false optiMoveSpeed=0.3 optiMoveAcceleration=0.09) feature=Base
    MoveDirectionNode (selectedDirection=ZPlus)
      Until TOOL_CONTACT_DETECTION (allowActions=false retraction=0 decelerationAcceleration=3 decelerationAngularAcceleration=34.906585)
  p3 := get_actual_tcp_pose()
  MoveJ speed 60 deg/s, acceleration 80 deg/s^2 (useActiveTCP=true optimoveEnabled=false optiMoveSpeed=0.3 optiMoveAcceleration=0.09) feature=Base
    Waypoint Variable (Variable): variable=ph7
    Waypoint Variable (Variable): variable=ph6
    Waypoint Waypoint_14: TCP in base x=-343.952 y=632.142 z=615.175 mm, rx=-0.0259 ry=-0.0088 rz=-0.5675 rad; joints [-77.363, -55.591, 142.791, -175.721, 90.298, 134.942] deg; TCP offset x=0 y=0 z=246 mm, rx=0 ry=0 rz=0 rad
    Waypoint Waypoint_4: TCP in base x=-658.265 y=299.53 z=30.91 mm, rx=0.4268 ry=-1.6215 rz=0.4371 rad; joints [-77.363, -55.591, 142.792, -102.186, -19.322, 105.94] deg
    Waypoint Waypoint_41: TCP in base x=392.128 y=533.269 z=644.149 mm, rx=0.0578 ry=2.126 rz=2.134 rad; joints [-198.126, -117.852, 133.303, -13.01, -11.421, -6.036] deg; TCP offset x=0 y=-4 z=284 mm, rx=0 ry=0 rz=0 rad
    'above waypoint is home'
  SuppressedNode
    SafeHome (positionOptionType=SPEED_AND_ACCELERATION speed=1.047198 acceleration=1.396263 nextMotionTime=2)
  ''
  ''
  ''
  ''
  ''
  ''
Thread Thread_1 (runOnlyOnce=true)
  Loop While (checkContinuously=false) expression=True
    If freedrive_m_var≟ True
      Script: freedrive_mode()
      free_dr_already := True
    Else 
      If free_dr_already
        Script: end_freedrive_mode()
    Script: sync()
SuppressedNode
  Thread Thread_2 (runOnlyOnce=false)
    Loop While (checkContinuously=false) expression=True
      If thread2trigger≟ True
        'do the dot extrude'
        Wait Sleep waitTime=5
        URCap WireTank Serial (WireTank Serial, WireTank, LLC) dataModel(byte_array=true, NODE_TITLE=Serial Bridge uR1, Command=[252,82,49], QUERY=false, OUTPUT_ENTRY=Static, Variable(key=OUTPUT_VARIABLE, variable(name=HwResp)))
        Wait Sleep waitTime=2
        URCap WireTank Serial (WireTank Serial, WireTank, LLC) dataModel(QUERY=false, NODE_TITLE=Serial Bridge uR0, Command=[252,82,48], byte_array=true, OUTPUT_ENTRY=Static, Variable(key=OUTPUT_VARIABLE, variable(name=HwResp)))
        thread2trigger := False
      Script: sync()
SubProgram move_path_3left (keepSynchronizedWithDisk=false) programFile=/programs/move_path_3left.urp
  'this is the path for Down, Over, then Back Around'
  ''
  MoveJ speed 60 deg/s, acceleration 80 deg/s^2 (useActiveTCP=true optimoveEnabled=false optiMoveSpeed=0.3 optiMoveAcceleration=0.09) feature=Base
    Waypoint Waypoint_37: TCP in base x=397.367 y=356.259 z=319.814 mm, rx=2.3163 ry=2.0576 rz=0.0741 rad; joints [-198.126, -117.852, 133.304, -13.009, -11.423, -6.036] deg; TCP offset x=-5.49 y=-328 z=106.39 mm, rx=1.2092 ry=-1.2092 rz=1.2092 rad
    'above point is home'
    Folder liftcolumnup
      liftcolumnz := liftcolumnzneeded
      If liftcolumnz>0
        URCap MachineLogic for Universal Robots (MachineLogic for Universal Robots, Vention Inc.) dataModel(type=addMotor, numberAdded=0, acceleration_in_mm_per_s2=50.0, ActuatorPos=liftcolumnz, speed_in_mm_per_min=3000.0, teachColor=BLUE, combo1=MachineMotion1, combo2=(1) Custom Actuator, combo3=Move to Position, combo6=In series, message=Move to Position, description=Moves the actuator to a specified position from the home location., comboAddress=Address 1, comboActuator=Valve 1)
    Waypoint Waypoint_15: TCP in base x=-157.621 y=513.354 z=815.678 mm, rx=-0.6727 ry=-1.8523 rz=-0.0554 rad; joints [-158.735, -104.322, 132.157, 58.275, -61.692, -46.244] deg; TCP offset x=-5.053 y=-331.71 z=103.574 mm, rx=1.2092 ry=-1.2092 rz=1.2092 rad
    Waypoint Waypoint_25: TCP in base x=-161.037 y=970.524 z=722.042 mm, rx=-0.555 ry=0.1065 rz=0.3286 rad; joints [-74.895, -76.586, 126.53, 213.07, -169.134, 52.325] deg; TCP offset x=-4.211 y=-279.829 z=105.916 mm, rx=1.2092 ry=-1.2092 rz=1.2092 rad
    Waypoint Waypoint_72: TCP in base x=-289.686 y=534.256 z=757.196 mm, rx=-0.2952 ry=-0.653 rz=0.3894 rad; joints [-79.881, -94.829, 156.625, 238.161, -217.62, 99.184] deg; TCP offset x=-5.49 y=-328 z=106.39 mm, rx=1.2092 ry=-1.2092 rz=1.2092 rad
    Waypoint Waypoint_26: TCP in base x=-689.651 y=138.963 z=230.691 mm, rx=-0.852 ry=-1.646 rz=1.646 rad; joints [-53.938, -86.03, 160.535, 285.425, -269.23, 90.049] deg; TCP offset x=-4.211 y=-279.829 z=105.916 mm, rx=1.2092 ry=-1.2092 rz=1.2092 rad
    Waypoint Waypoint_27: TCP in base x=-568.725 y=230.602 z=220.208 mm, rx=-1.5191 ry=-0.5352 rz=0.574 rad; joints [-2.798, -73.075, 141.93, 288.829, -133.322, 87.786] deg; TCP offset x=8.385 y=-333.249 z=78.524 mm, rx=1.2092 ry=-1.2092 rz=1.2092 rad
    SuppressedNode
      Waypoint Waypoint_1: TCP in base x=-1177.596 y=138.956 z=230.69 mm, rx=-0.852 ry=-1.646 rz=1.646 rad; joints [-20.637, -63.427, 120.718, 302.664, -235.94, 90.036] deg; TCP offset x=-4.211 y=-279.829 z=105.916 mm, rx=1.2092 ry=-1.2092 rz=1.2092 rad
    SuppressedNode
      Waypoint Waypoint_2: TCP in base x=-689.651 y=138.963 z=230.691 mm, rx=-0.852 ry=-1.646 rz=1.646 rad; joints [-53.938, -86.03, 160.535, 285.425, -269.23, 90.049] deg
    SuppressedNode
      Waypoint Waypoint_3: TCP in base x=-161.037 y=970.524 z=722.042 mm, rx=-0.555 ry=0.1065 rz=0.3286 rad; joints [-74.895, -76.586, 126.53, 213.07, -169.134, 52.325] deg
    SuppressedNode
      SafeHome (positionOptionType=SPEED_AND_ACCELERATION speed=1.047198 acceleration=1.396263 nextMotionTime=2)
  ''
  p1 := pathturn[0]
  p2 := pathturn[1]
  p4 := pathturn[2]
  p5 := pathturn[3]
  pa1 := p[p1[0]+0.05,p1[1]-0.05,p1[2],p1[3],p1[4],p1[5]]
  MoveJ speed 60 deg/s, acceleration 80 deg/s^2 (useActiveTCP=true optimoveEnabled=false optiMoveSpeed=0.3 optiMoveAcceleration=0.09) feature=Base
    Waypoint Variable (Variable): variable=pa1
  MoveL speed 50 mm/s, acceleration 100 mm/s^2 (useActiveTCP=true optimoveEnabled=false optiMoveSpeed=0.3 optiMoveAcceleration=0.09) feature=Base
    Waypoint Variable (Variable): variable=p1
  Wait Sleep waitTime=8
  URCap WireTank Serial (WireTank Serial, WireTank, LLC) dataModel(NODE_TITLE=Serial Bridge uR1, Command=[252,82,49], byte_array=true, OUTPUT_ENTRY=Static)
  URCap WireTank Serial (WireTank Serial, WireTank, LLC) dataModel(NODE_TITLE=Serial Bridge uR1, Command=[252,82,49], QUERY=false, byte_array=true, OUTPUT_ENTRY=Static, Variable(key=OUTPUT_VARIABLE, variable(name=HwResp)))
  Wait Sleep waitTime=1
  SuppressedNode
    Script: turn_extrusion_on()
  Set DigitalOutput pin=digital_out[0]; digitalValue=1
  MoveL speed 10 mm/s, acceleration 100 mm/s^2 (useActiveTCP=true optimoveEnabled=false optiMoveSpeed=0.3 optiMoveAcceleration=0.09) feature=Base
    Waypoint Variable (Variable): variable=p2
  URCap WireTank Serial (WireTank Serial, WireTank, LLC) dataModel(NODE_TITLE=Serial Bridge uR0, byte_array=true, Command=[252,82,48], OUTPUT_ENTRY=Static)
  Wait Sleep waitTime=0.5
  Set DigitalOutput pin=digital_out[0]; digitalValue=0
  MoveL speed 120 mm/s, acceleration 10 mm/s^2 (useActiveTCP=true optimoveEnabled=false optiMoveSpeed=0.3 optiMoveAcceleration=0.09) feature=Base
    Waypoint Variable (Variable): variable=p4
  URCap WireTank Serial (WireTank Serial, WireTank, LLC) dataModel(NODE_TITLE=Serial Bridge uR1, byte_array=true, Command=[252,82,49], OUTPUT_ENTRY=Static)
  URCap WireTank Serial (WireTank Serial, WireTank, LLC) dataModel(NODE_TITLE=Serial Bridge uR1, Command=[252,82,49], QUERY=false, byte_array=true, OUTPUT_ENTRY=Static, Variable(key=OUTPUT_VARIABLE, variable=HwResp))
  Wait Sleep waitTime=1
  SuppressedNode
    Script: turn_extrusion_on()
  Set DigitalOutput pin=digital_out[0]; digitalValue=1
  MoveL speed 10 mm/s, acceleration 100 mm/s^2 (useActiveTCP=true optimoveEnabled=false optiMoveSpeed=0.3 optiMoveAcceleration=0.09) feature=Base
    Waypoint Variable (Variable): variable=p5
  URCap WireTank Serial (WireTank Serial, WireTank, LLC) dataModel(NODE_TITLE=Serial Bridge uR0, Command=[252,82,48], byte_array=true, OUTPUT_ENTRY=Static)
  Wait Sleep waitTime=2
  Set DigitalOutput pin=digital_out[0]; digitalValue=0
  ''
  pret1 := p[p5[0]+.1,p5[1],p5[2],p5[3],p5[4],p5[5]]
  p_1 := pathturn[4]
  p_2 := pathturn[5]
  p_3 := pathturn[6]
  p_4 := pathturn[7]
  p_5 := pathturn[8]
  p_preheat := p[p_3[0]+.01,p_3[1],p_3[2],p_3[3],p_3[4],p_3[5]]
  p_pre_ret := p[p_1[0]+.03,p_1[1]-.03,p_1[2],p_1[3],p_1[4],p_1[5]]
  p_pre_ret2 := p[p_3[0]+.03,p_3[1],p_3[2],p_3[3],p_3[4],p_3[5]]
  MoveJ speed 80 deg/s, acceleration 80 deg/s^2 (useActiveTCP=true optimoveEnabled=false optiMoveSpeed=0.3 optiMoveAcceleration=0.09) feature=Base
    Waypoint Variable (Variable): variable=pret1
    Waypoint Waypoint_28: TCP in base x=-568.725 y=230.602 z=220.208 mm, rx=-1.5191 ry=-0.5352 rz=0.574 rad; joints [-2.798, -73.075, 141.93, 288.829, -133.322, 87.786] deg; TCP offset x=8.385 y=-333.249 z=78.524 mm, rx=1.2092 ry=-1.2092 rz=1.2092 rad
    If liftcolumnz≠0.0
      URCap MachineLogic for Universal Robots (MachineLogic for Universal Robots, Vention Inc.) dataModel(type=addMotor, numberAdded=0, speed_in_mm_per_min=600, acceleration_in_mm_per_s2=50.0, teachColor=BLUE, combo1=MachineMotion1, combo2=(1) Custom Actuator, combo3=Home, combo6=In series, message=Homing, description=Moves the actuator in the negative direction until the home sensor is triggered and sets position to zero (0)., comboAddress=Address 1, comboActuator=Valve 1)
    'now go into the ccw weld position'
    Waypoint Waypoint_29: TCP in base x=-689.651 y=138.963 z=230.691 mm, rx=-0.852 ry=-1.646 rz=1.646 rad; joints [-53.938, -86.03, 160.535, 285.425, -269.23, 90.049] deg; TCP offset x=-4.211 y=-279.829 z=105.916 mm, rx=1.2092 ry=-1.2092 rz=1.2092 rad
    ''
    Waypoint Waypoint_30: TCP in base x=-853.851 y=133.267 z=60.418 mm, rx=-0.2742 ry=-2.3597 rz=0.0468 rad; joints [-34.868, -57.997, 159.687, 213.62, -283.084, 21.643] deg; TCP offset x=8.385 y=-333.249 z=78.524 mm, rx=1.2092 ry=-1.2092 rz=1.2092 rad
    Waypoint Waypoint_31: TCP in base x=-979.398 y=-259.625 z=211.289 mm, rx=-0.673 ry=-1.4594 rz=-0.6402 rad; joints [21.182, -32.844, 122.516, 179.072, -269.511, -69.331] deg
    SuppressedNode
      Waypoint Waypoint_9: TCP in base x=-161.037 y=970.524 z=722.042 mm, rx=-0.555 ry=0.1065 rz=0.3286 rad; joints [-74.895, -76.586, 126.53, 213.07, -169.134, 52.325] deg; TCP offset x=-4.211 y=-279.829 z=105.916 mm, rx=1.2092 ry=-1.2092 rz=1.2092 rad
    SuppressedNode
      Waypoint Waypoint_22: TCP in base x=-308.534 y=606.085 z=242.393 mm, rx=1.3699 ry=1.0669 rz=-1.2572 rad; joints [-84.142, -55.374, 92.791, 53.186, 94.965, 15.074] deg
  SuppressedNode
    MoveP speed 20 mm/s, acceleration 2 mm/s^2 (blendRadius=0.001 useActiveTCP=true optimoveEnabled=false optiMoveSpeed=0.3 optiMoveAcceleration=0.09) feature=Base
      'below (until next comment) are points for testing out ccw circle weld'
      Waypoint Waypoint_8: TCP in base x=-1291.697 y=90.422 z=23.176 mm, rx=-0.673 ry=-1.4594 rz=-0.6402 rad; joints [-2.307, -18.609, 101.914, 185.717, -269.053, -45.852] deg; TCP offset x=8.385 y=-333.249 z=78.524 mm, rx=1.2092 ry=-1.2092 rz=1.2092 rad
      Waypoint Waypoint_10: TCP in base x=-1193.179 y=196.591 z=23.164 mm, rx=-0.673 ry=-1.4594 rz=-0.6402 rad; joints [-8.888, -18.95, 110.853, 177.226, -268.954, -39.273] deg
      Waypoint Waypoint_11: TCP in base x=-1193.173 y=196.572 z=23.158 mm, rx=0.078 ry=-1.5698 rz=0.1134 rad; joints [-28.391, -18.785, 116.78, 172.699, -268.884, 35.453] deg
      'end test points'
  MoveL speed 250 mm/s, acceleration 1200 mm/s^2 (useActiveTCP=true optimoveEnabled=false optiMoveSpeed=0.3 optiMoveAcceleration=0.09) feature=Base
    Waypoint Variable (Variable): variable=p_pre_ret
    Waypoint Variable (Variable): variable=p_pre_ret2
    Waypoint Variable (Variable): variable=p_preheat
  Wait Sleep waitTime=6
  MoveL speed 250 mm/s, acceleration 1200 mm/s^2 (useActiveTCP=true optimoveEnabled=false optiMoveSpeed=0.3 optiMoveAcceleration=0.09) feature=Base
    Waypoint Variable (Variable): variable=p_pre_ret2
    Waypoint Variable (Variable): variable=p_pre_ret
  Set NoAction tcp=backofhole
  MoveL speed 50 mm/s, acceleration 100 mm/s^2 (useActiveTCP=true optimoveEnabled=false optiMoveSpeed=0.3 optiMoveAcceleration=0.09) feature=Base
    Waypoint Variable (Variable): variable=p_1
  URCap WireTank Serial (WireTank Serial, WireTank, LLC) dataModel(NODE_TITLE=Serial Bridge uR1, Command=[252,82,49], OUTPUT_ENTRY=Static, byte_array=true)
  URCap WireTank Serial (WireTank Serial, WireTank, LLC) dataModel(NODE_TITLE=Serial Bridge uR1, Command=[252,82,49], QUERY=false, byte_array=true, OUTPUT_ENTRY=Static, Variable(key=OUTPUT_VARIABLE, variable(name=HwResp)))
  Wait Sleep waitTime=1
  Set DigitalOutput pin=digital_out[0]; digitalValue=1
  SuppressedNode
    Script: turn_extrusion_on()
  Wait Sleep waitTime=1
  MoveL speed 10 mm/s, acceleration 1200 mm/s^2 (useActiveTCP=true optimoveEnabled=false optiMoveSpeed=0.3 optiMoveAcceleration=0.09) feature=Base
    Waypoint Variable (Variable): variable=p_2
  MoveP speed 0.5 mm/s, acceleration 10 mm/s^2 (blendRadius=0.001 useActiveTCP=true optimoveEnabled=false optiMoveSpeed=0.3 optiMoveAcceleration=0.09) feature=Base
    CircleMove (OrientationMode=FIXED)
      Waypoint Variable (Variable): variable=p_3
      Waypoint Variable (Variable): variable=p_4
  MoveL speed 12 mm/s, acceleration 1200 mm/s^2 (useActiveTCP=true optimoveEnabled=false optiMoveSpeed=0.3 optiMoveAcceleration=0.09) feature=Base
    Waypoint Variable (Variable): variable=p_5
  URCap WireTank Serial (WireTank Serial, WireTank, LLC) dataModel(NODE_TITLE=Serial Bridge uR0, Command=[252,82,48], byte_array=true, OUTPUT_ENTRY=Static)
  Wait Sleep waitTime=2
  Set DigitalOutput pin=digital_out[0]; digitalValue=0
  SuppressedNode
    MoveL speed 250 mm/s, acceleration 1200 mm/s^2 (useActiveTCP=true optimoveEnabled=false optiMoveSpeed=0.3 optiMoveAcceleration=0.09) feature=Base
      Waypoint Waypoint_23: TCP in base x=-540.167 y=215.949 z=34.631 mm, rx=-1.5058 ry=1.0576 rz=1.5735 rad; joints [-26.452, -65.119, 143.749, 8.723, 85.674, 218.843] deg; TCP offset x=-4.211 y=-279.829 z=105.916 mm, rx=1.2092 ry=-1.2092 rz=1.2092 rad
  SuppressedNode
    MoveJ speed 60 deg/s, acceleration 80 deg/s^2 (useActiveTCP=true optimoveEnabled=false optiMoveSpeed=0.3 optiMoveAcceleration=0.09) feature=Base
      Waypoint Waypoint_24: TCP in base x=-308.526 y=606.096 z=242.373 mm, rx=-2.1337 ry=0.3494 rz=2.1309 rad; joints [-107.196, -73.784, 125.643, 43.029, 90.975, 86.468] deg
  MoveJ speed 60 deg/s, acceleration 80 deg/s^2 (useActiveTCP=true optimoveEnabled=false optiMoveSpeed=0.3 optiMoveAcceleration=0.09) feature=Base
    Waypoint Waypoint_32: TCP in base x=-826.866 y=369.358 z=43.114 mm, rx=0.575 ry=-1.4922 rz=0.5971 rad; joints [-59.333, -19.441, 121.825, 168.37, -269.932, 102.332] deg; TCP offset x=8.385 y=-333.249 z=78.524 mm, rx=1.2092 ry=-1.2092 rz=1.2092 rad
    Waypoint Waypoint_33: TCP in base x=-689.651 y=138.963 z=230.691 mm, rx=-0.852 ry=-1.646 rz=1.646 rad; joints [-53.938, -86.03, 160.535, 285.425, -269.23, 90.049] deg; TCP offset x=-4.211 y=-279.829 z=105.916 mm, rx=1.2092 ry=-1.2092 rz=1.2092 rad
    Waypoint Waypoint_73: TCP in base x=-289.671 y=534.275 z=757.233 mm, rx=-0.2952 ry=-0.653 rz=0.3894 rad; joints [-79.881, -94.83, 156.622, 238.16, -217.619, 99.184] deg; TCP offset x=-5.49 y=-328 z=106.39 mm, rx=1.2092 ry=-1.2092 rz=1.2092 rad
  ''
  MoveJ speed 60 deg/s, acceleration 80 deg/s^2 (useActiveTCP=true optimoveEnabled=false optiMoveSpeed=0.3 optiMoveAcceleration=0.09) feature=Base
    Waypoint Waypoint_16: TCP in base x=191.113 y=567.512 z=815.514 mm, rx=-0.1358 ry=0.3961 rz=0.2088 rad; joints [-94.746, -100.957, 150.262, 188.452, -152.118, 48.82] deg; TCP offset x=-5.053 y=-331.71 z=103.574 mm, rx=1.2092 ry=-1.2092 rz=1.2092 rad
    Waypoint Waypoint_17: TCP in base x=-254.566 y=502.963 z=1135.402 mm, rx=-0.2619 ry=-0.7497 rz=1.349 rad; joints [-116.61, -108.45, 141.427, 125.702, -66.866, -29.172] deg
    Waypoint Waypoint_18: TCP in base x=-9.208 y=593.718 z=505.81 mm, rx=-1.4244 ry=-2.3441 rz=-0.5276 rad; joints [-167.145, -114.278, 136.39, 39.71, -32.494, -66.269] deg
    Waypoint Waypoint_38: TCP in base x=397.38 y=356.252 z=319.817 mm, rx=2.3163 ry=2.0576 rz=0.0741 rad; joints [-198.126, -117.852, 133.304, -13.01, -11.422, -6.036] deg; TCP offset x=-5.49 y=-328 z=106.39 mm, rx=1.2092 ry=-1.2092 rz=1.2092 rad
    'above point is home'
